Fanuc KAREL source: KA00196.KL

PROGRAM KA00196
%NOLOCKGROUP
VAR
  SRC: ARRAY[4] OF SHORT
  DST: ARRAY[4] OF VECTOR
BEGIN
  DST = SRC
END KA00196
